TYPE TcoDatamanResultsControl_v_5_x_x : 
STRUCT
    EnableResultBuffering AT %Q* : BOOL;
    ResultsAcknowledge AT %Q* : BOOL;
END_STRUCT
END_TYPE

(* stored: Version 1.1.0.1, ProductVersion 3.1.4024.11
   DUT TcoDatamanResultsControl_v_5_x_x: Id {71ac6516-8a2f-4944-806f-469cb653cd56} *)
